(* CoDeSys 2.3.5.6 project: szlendak_03_LD.pro *)
(* Libraries: Standard.lib 31.10.14 11:17:58, SYSLIBCALLBACK.LIB 31.10.14 11:17:58 *)

(* PLC configuration (modules and I/O channels)
Configuration EC4P-200 [Root] node -1, in %IB0 out %QB0 {EC4P_RestartPwrOn = WARMSTART; EC4P_MaxCycleTime = 20; EC4P_Com1BaudRate = 38400; EC4P_CAN1BaudRate = 125KBaud; EC4P_RoutingId = 127; EC4P_EasyNetId = 1; EC4P_EasyNetCfg = 0; EC4P_EasyNetCycleTime = 50; EC4P_RoutingChannel = CAN1; EC4P_IPFlags = 0; EC4P_IPAddress = 0; EC4P_SubNetMask = 0; EC4P_DefaultGateway = 0; EC4P_SummerWinterFlags = 0; EC4P_SummerWinterRule1 = 0; EC4P_SummerWinterRule2 = 0}
  Local I/O [EC4P_LocalIO] node 0, in %IB0 out %QB0 {EC4P_LocalInt = 0}
    I1 AT %IX0.0 [LocalBitInput] Input I1
    I2 AT %IX0.1 [LocalBitInput] Input I2
    I3 AT %IX0.2 [LocalBitInput] Input I3
    I4 AT %IX0.3 [LocalBitInput] Input I4
    I5 AT %IX0.4 [LocalBitInput] Input I5
    I6 AT %IX0.5 [LocalBitInput] Input I6
    I7 AT %IX0.6 [LocalBitInput] Input I7
    I8 AT %IX0.7 [LocalBitInput] Input I8
    I9 AT %IX1.0 [LocalBitInput] Input I9
    I10 AT %IX1.1 [LocalBitInput] Input I10
    I11 AT %IX1.2 [LocalBitInput] Input I11
    I12 AT %IX1.3 [LocalBitInput] Input I12
    I13 AT %IX1.4 [LocalDiagInput] Diagnostic Input I13
    I14 AT %IX1.5 [LocalDiagInput] Diagnostic Input I14
    I15 AT %IX1.6 [LocalDiagInput] Diagnostic Input I15
    I16 AT %IX1.7 [LocalDiagInput] Diagnostic Input I16
    I7_Analog AT %IW2 [LocalAnalogIn] Input I7, 10Bit, 0-10VDC
    I8_Analog AT %IW4 [LocalAnalogIn] Input I8, 10Bit, 0-10VDC
    I11_Analog AT %IW6 [LocalAnalogIn] Input I11, 10Bit, 0-10VDC
    I12_Analog AT %IW8 [LocalAnalogIn] Input I12, 10Bit, 0-10VDC
    Transistor Outputs [EC4P_TOutputs] node 0, in %IB10 out %QB0
      Q1 AT %QX0.0 [LocalBitOutput] Transistor-Output Q1
      Q2 AT %QX0.1 [LocalBitOutput] Transistor-Output Q2
      Q3 AT %QX0.2 [LocalBitOutput] Transistor-Output Q3
      Q4 AT %QX0.3 [LocalBitOutput] Transistor-Output Q4
      Q5 AT %QX0.4 [LocalBitOutput] Transistor-Output Q5
      Q6 AT %QX0.5 [LocalBitOutput] Transistor-Output Q6
      Q7 AT %QX0.6 [LocalBitOutput] Transistor-Output Q7
      Q8 AT %QX0.7 [LocalBitOutput] Transistor-Output Q8
    No Analog Output [EC4P_NoAnalogOutput] node 1, in %IB10 out %QB1
    No Keys [EC4P_NoKeys] node 2, in %IB10 out %QB1
    No Counter [EC4P_NoCounter] node 3, in %IB10 out %QB1
  Extension [EC4P_Extension] node 1, in %IB10 out %QB1
    No Extension [EC4P_NoExtension] node 0, in %IB10 out %QB1
*)

(* POU PLC_PRG, LD *)
PROGRAM PLC_PRG
VAR
	CTU_3: CTU;
	LICZBA: INT;
	RESET: BOOL;
	TP_1: TP;
	T_TP_1: TIME;
	L1: BOOL;
	TON_1: TON;
	T_TON_1: TIME;
	CU: BOOL;
	TON_2: TON;
	T_TON_2: TIME;
	Y1: BOOL;
	Y2: BOOL;
	Y3: BOOL;
	Y4: BOOL;
	Y5: BOOL;
	Y6: BOOL;
	Y7: BOOL;
	Y8: BOOL;
	Y9: BOOL;
	Y0: BOOL;
END_VAR
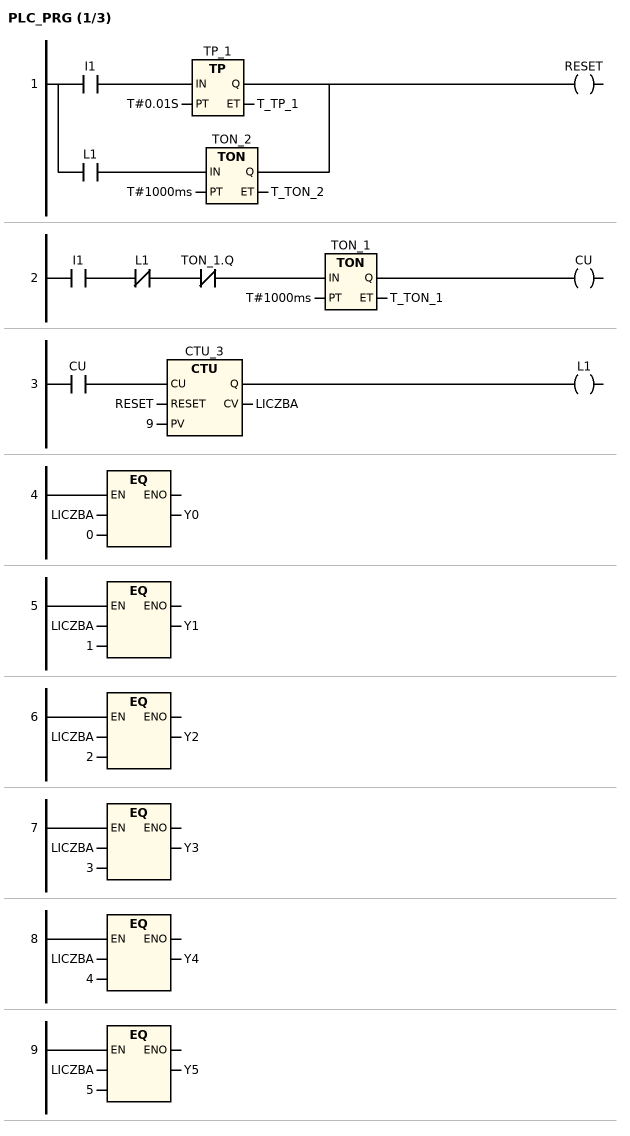
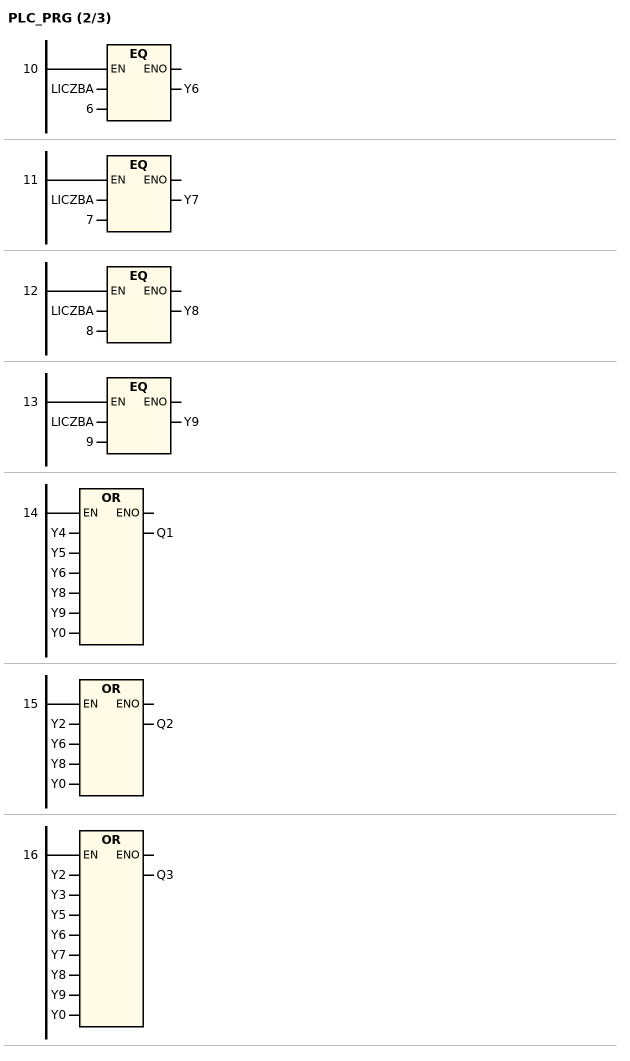
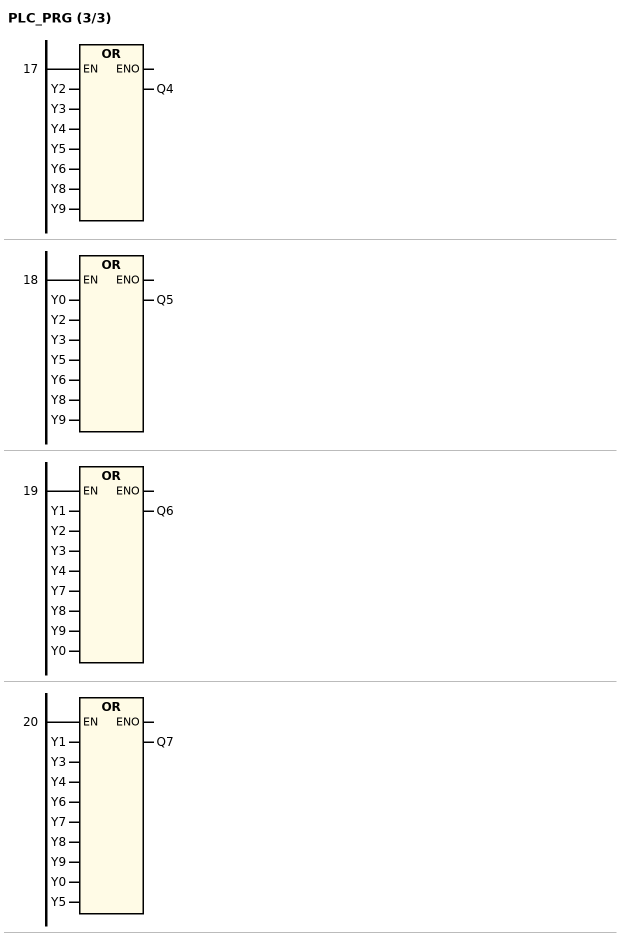
_LD_ (* Ladder Diagram *)
NETWORK 1
	{ [I1] - TP_1:TP(IN: *, PT: T#0.01S, ET => T_TP_1) | [L1] - TON_2:TON(IN: *, PT: T#1000ms, ET => T_TON_2) } --- (RESET)
NETWORK 2
	[I1] - [/L1] - [/TON_1.Q] - TON_1:TON(IN: *, PT: T#1000ms, ET => T_TON_1) --- (CU)
NETWORK 3
	[CU] - CTU_3:CTU(CU: *, RESET: RESET, PV: 9, CV => LICZBA) --- (L1)
NETWORK 4
	*
		EN --- EQ(LICZBA, 0) => Y0
NETWORK 5
	*
		EN --- EQ(LICZBA, 1) => Y1
NETWORK 6
	*
		EN --- EQ(LICZBA, 2) => Y2
NETWORK 7
	*
		EN --- EQ(LICZBA, 3) => Y3
NETWORK 8
	*
		EN --- EQ(LICZBA, 4) => Y4
NETWORK 9
	*
		EN --- EQ(LICZBA, 5) => Y5
NETWORK 10
	*
		EN --- EQ(LICZBA, 6) => Y6
NETWORK 11
	*
		EN --- EQ(LICZBA, 7) => Y7
NETWORK 12
	*
		EN --- EQ(LICZBA, 8) => Y8
NETWORK 13
	*
		EN --- EQ(LICZBA, 9) => Y9
NETWORK 14
	*
		EN --- OR(Y4, Y5, Y6, Y8, Y9, Y0) => Q1
NETWORK 15
	*
		EN --- OR(Y2, Y6, Y8, Y0) => Q2
NETWORK 16
	*
		EN --- OR(Y2, Y3, Y5, Y6, Y7, Y8, Y9, Y0) => Q3
NETWORK 17
	*
		EN --- OR(Y2, Y3, Y4, Y5, Y6, Y8, Y9) => Q4
NETWORK 18
	*
		EN --- OR(Y0, Y2, Y3, Y5, Y6, Y8, Y9) => Q5
NETWORK 19
	*
		EN --- OR(Y1, Y2, Y3, Y4, Y7, Y8, Y9, Y0) => Q6
NETWORK 20
	*
		EN --- OR(Y1, Y3, Y4, Y6, Y7, Y8, Y9, Y0, Y5) => Q7
_END_LD_
(* the same logic as Structured Text *)
(* Network 1 *)
TP_1(IN := I1, PT := T#0.01S);
T_TP_1 := TP_1.ET;
TON_2(IN := L1, PT := T#1000ms);
T_TON_2 := TON_2.ET;
RESET := TP_1.Q OR TON_2.Q;
(* Network 2 *)
TON_1(IN := I1 AND NOT L1 AND NOT TON_1.Q, PT := T#1000ms);
T_TON_1 := TON_1.ET;
CU := TON_1.Q;
(* Network 3 *)
CTU_3(CU := CU, RESET := RESET, PV := 9);
LICZBA := CTU_3.CV;
L1 := CTU_3.Q;
(* Network 4 *)
Y0 := LICZBA = 0;
(* Network 5 *)
Y1 := LICZBA = 1;
(* Network 6 *)
Y2 := LICZBA = 2;
(* Network 7 *)
Y3 := LICZBA = 3;
(* Network 8 *)
Y4 := LICZBA = 4;
(* Network 9 *)
Y5 := LICZBA = 5;
(* Network 10 *)
Y6 := LICZBA = 6;
(* Network 11 *)
Y7 := LICZBA = 7;
(* Network 12 *)
Y8 := LICZBA = 8;
(* Network 13 *)
Y9 := LICZBA = 9;
(* Network 14 *)
Q1 := Y4 OR Y5 OR Y6 OR Y8 OR Y9 OR Y0;
(* Network 15 *)
Q2 := Y2 OR Y6 OR Y8 OR Y0;
(* Network 16 *)
Q3 := Y2 OR Y3 OR Y5 OR Y6 OR Y7 OR Y8 OR Y9 OR Y0;
(* Network 17 *)
Q4 := Y2 OR Y3 OR Y4 OR Y5 OR Y6 OR Y8 OR Y9;
(* Network 18 *)
Q5 := Y0 OR Y2 OR Y3 OR Y5 OR Y6 OR Y8 OR Y9;
(* Network 19 *)
Q6 := Y1 OR Y2 OR Y3 OR Y4 OR Y7 OR Y8 OR Y9 OR Y0;
(* Network 20 *)
Q7 := Y1 OR Y3 OR Y4 OR Y6 OR Y7 OR Y8 OR Y9 OR Y0 OR Y5;
END_PROGRAM

(* POU counter_cfc, CFC *)
PROGRAM counter_cfc
VAR
END_VAR
_CFC_ (* Continuous Function Chart, elements in execution order *)
_END_CFC_
END_PROGRAM
